TYPE ST_PlanarTrackConfig :
STRUCT
	TrackIndex					: E_TrackNum;
	MCTrack						: CDT_MCTOPLC_PLANAR_TRACK;
END_STRUCT
END_TYPE

(* stored: Version 1.1.0.1, ProductVersion 3.1.4026.8
   DUT ST_PlanarTrackConfig: Id {41fd4cc1-ca39-0eac-1ee8-d3be3f06a63e} *)
